FUNCTION_BLOCK A2X2_2X_TO_BOOL (* Composite FB for convert A2X2 to 2 BOOLS *)
  (* Standard: 61499-2; Description: Copyright (c) 2026 HR Agrartechnik GmbH This program and the accompanying materials are made available under the terms of the Eclipse Public License 2.0 which is available at https://www.eclipse.org/legal/epl-2.0/ SPDX-License-Identifier: EPL-2.0 *)
  (* Version 1.0, 2026-08-31, Franz Höpfinger, HR Agrartechnik GmbH *)
  PACKAGE adapter::conversion::bidirectional;
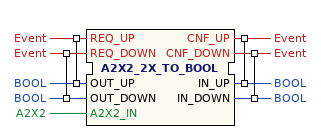
  EVENT_INPUT
    REQ_UP WITH OUT_UP; (* Request UP to Adapter *)
    REQ_DOWN WITH OUT_DOWN; (* Request DOWN to Adapter *)
  END_EVENT
  EVENT_OUTPUT
    CNF_UP WITH IN_UP; (* Confirmation UP from Adapter *)
    CNF_DOWN WITH IN_DOWN; (* Confirmation DOWN from Adapter *)
  END_EVENT
  VAR_INPUT
    OUT_UP : BOOL; (* TRUE = forward, up, right, clockwise *)
    OUT_DOWN : BOOL; (* TRUE = backward, down, left, counter-clockwise *)
  END_VAR
  VAR_OUTPUT
    IN_UP : BOOL; (* UP data from Adapter *)
    IN_DOWN : BOOL; (* DOWN data from Adapter *)
  END_VAR
  SOCKETS
    A2X2_IN : adapter::types::bidirectional::A2X2; (* Adapter Input *)
  END_SOCKETS
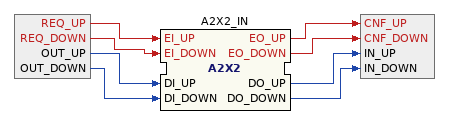
  EVENT_CONNECTIONS
    A2X2_IN.EO_UP TO CNF_UP;
    A2X2_IN.EO_DOWN TO CNF_DOWN;
    REQ_UP TO A2X2_IN.EI_UP;
    REQ_DOWN TO A2X2_IN.EI_DOWN;
  END_CONNECTIONS
  DATA_CONNECTIONS
    A2X2_IN.DO_UP TO IN_UP;
    A2X2_IN.DO_DOWN TO IN_DOWN;
    OUT_UP TO A2X2_IN.DI_UP;
    OUT_DOWN TO A2X2_IN.DI_DOWN;
  END_CONNECTIONS
END_FUNCTION_BLOCK
